{attribute addProperty BoxType "EL2262-0000-0001"}
{attribute addProperty Id "Output0AT %Q*BOOL81"}
{attribute addProperty CRC "2885009065"}
{attribute addProperty SizeInBites "8"}
{attribute addProperty SizeInBytes "1"}
TYPE Sample_ABF5BEA9 :
STRUCT
	{attribute addProperty Name "Output0"}
	Output0 AT %Q* : BOOL;
END_STRUCT
END_TYPE

(* stored: Version 1.2.0.0, ProductVersion 3.1.4024.9
   DUT Sample_ABF5BEA9: Id {295849aa-6468-4fb0-bddd-474cddc4e697} *)
